{attribute 'qualified_only'}
{attribute 'strict'}
{attribute 'to_string'}
TYPE eSkillCommandType :
(
    None    := 0,
    Start   := 1,
    Stop    := 2,
    Abort   := 3,
    Restart := 4
);
END_TYPE

(* stored: Version 1.1.0.1, ProductVersion 3.1.4026.18
   DUT eSkillCommandType: Id {55711a49-414b-4e06-a38e-ba422bc9de0d} *)
